SUBAPPLICATION Uebung_Interlock_AX (* Interlock advanced exercise (AX) *)
  (* Standard: 61499-2; Description: Copyright (c) 2026 Meisterschulen am Ostbahnhof *)
  (* Version 1.0, 2026-05-07, Gemini CLI, Meisterschulen am Ostbahnhof, Interlock exercise *)
  PACKAGE Uebungen;
  IMPORT logiBUS::signalprocessing::interlock::ILOCK_IO_AX;
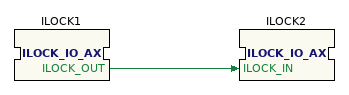
  FBS
    ILOCK1 : logiBUS::signalprocessing::interlock::ILOCK_IO_AX;
    ILOCK2 : logiBUS::signalprocessing::interlock::ILOCK_IO_AX;
  END_FBS
  ADAPTER_CONNECTIONS
    ILOCK1.ILOCK_OUT TO ILOCK2.ILOCK_IN;
  END_CONNECTIONS
END_SUBAPPLICATION
